// TIA Portal project "Gluing_A1" (V13)

(* hardware
DEVICE "S7300/ET200M-Station_1"  S7-300 station
   slot 0: "Profilschiene_0"  Rail  6ES7 390-1***0-0AA0
   slot 1: "PS 307 5A_1"  PS 307 5A  6ES7 307-1EA00-0AA0
   slot 2: "SIMATIC S7-300"  CPU 314C-2 PN/DP  6ES7 314-6EH04-0AB0  V3.3
      slot 2: "PROFINET-Schnittstelle_1"  PN-IO
         slot 1: "Port_1"  Port
         slot 2: "Port_2"  Port
      slot 5: "DI 24/DO 16_1"  DI24/DO16
      slot 6: "AI 5/AO 2_1"  AI5/AO2
      slot 7: "Zählen_1"  Counter
      slot 8: "Positionieren_1"  Positioning
   slot 4: "CP 343-2_1"  CP 343-2  6GK7 343-2AH01-0XA0  V3.1
*)

// ===== PLC "SIMATIC S7-300"  CPU 314C-2 PN/DP =====

VAR_GLOBAL   // PLC tag table "Standard-Variablentabelle"
   "Ix_S1_Start" AT %I124.0 : Bool;   // Start Pushbutton 1
   "Ix_S2_Start" AT %I124.1 : Bool;   // Start Pushbutton 2
   "Ix_1B1_PressCyl1A1Ret" AT %I124.2 : Bool;   // Press Cylinder 1A1 retracted
   "Ix_1B2_PressCyl1A1Ext" AT %I124.3 : Bool;   // Press Cylinder 1A1 extended
   "Qx_1M1_MovePressCyl1A1Out" AT %Q124.0 : Bool;   // Move PressCylinder 1A1 out
   "Qx_P1_GluingProcess" AT %Q124.7 : Bool;   // Signalise the gluing process
   "Mb_FlagByte10" AT %MB10 : Byte;   // Flag byte 10
   "Mx_Step0" AT %M10.0 : Bool;   // Grafcet, step-flag 0
   "Mx_Step1" AT %M10.1 : Bool;   // Grafcet, step-flag1
   "Mx_Step2" AT %M10.2 : Bool;   // Grafcet, step-flag2
   "Mx_Step3" AT %M10.3 : Bool;   // Grafcet, step-flag3
   "Mx_Step4" AT %M10.4 : Bool;   // Grafcet, step-flag4
   "Mx_Step5" AT %M10.5 : Bool;   // Grafcet, step-flag5
   "Mx_Step6" AT %M10.6 : Bool;   // Grafcet, step-flag6
   "Mx_StartingFlag" AT %M20.0 : Bool;   // Starting flag to activate the sequence (Step 0)
   "Mx_NEdegFlag_Step2" AT %M20.1 : Bool;   // Negative edge flag is activated wehn step 2 is deactivated
   "Mx_Clock10Hz" AT %M100.0 : Bool;   // CPU clock memory-flag 0:f = 10Hz / T=0,1s
   "Mx_Clock5Hz" AT %M100.1 : Bool;   // CPU clock memory-flag 1:f = 5Hz / T=0,2s
   "Mx_Clock2,5Hz" AT %M100.2 : Bool;   // CPU clock memory-flag 2:f = 2,5Hz / T=0,4s
   "Mx_Clock2Hz" AT %M100.3 : Bool;   // CPU clock memory-flag 3:f = 2Hz / T=0,5s
   "Mx_Clock1,2Hz" AT %M100.4 : Bool;   // CPU clock memory-flag 4:f = 1,2Hz / T=0,8s
   "Mx_Clock1Hz" AT %M100.5 : Bool;   // CPU clock memory-flag 5:f = 1Hz / T=1s
   "Mx_Clock0,65Hz" AT %M100.6 : Bool;   // CPU clock memory-flag 6:f = 0,65Hz / T=1,6s
   "Mx_Clock0,5Hz" AT %M100.7 : Bool;   // CPU clock memory-flag 7:f = 0,5Hz / T=2s
   "T_GlueTime" AT %T1 : Timer;   // Adjusting the gluing time
END_VAR

DATA_BLOCK "gluning time value"   // DB2
{ S7_Optimized_Access := 'FALSE' }
VERSION : 0.1
   VAR
      "GluingValue Siemens" : S5Time;
      "GluingValue ICE" : Time;
   END_VAR
BEGIN
END_DATA_BLOCK

FUNCTION "Grafecet" : Void   // FC1, FBD
{ S7_Optimized_Access := 'FALSE' }
VERSION : 0.1
BEGIN

REGION Network 1: step 0
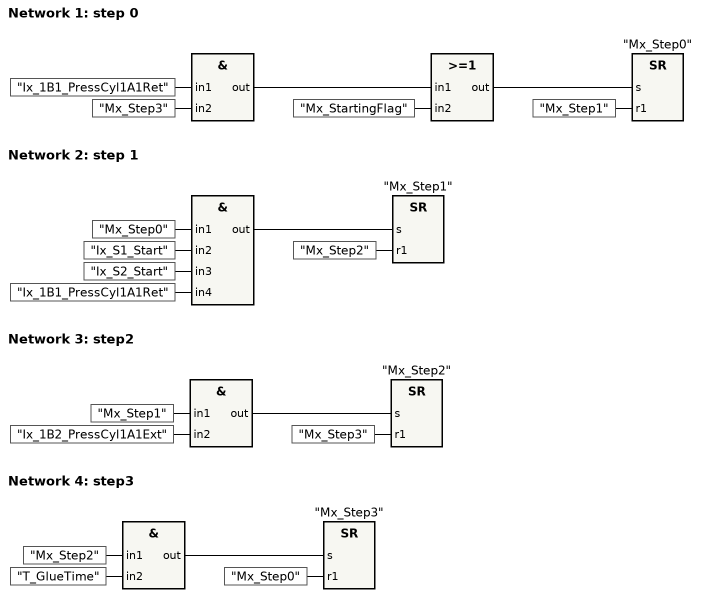
   IF ("Ix_1B1_PressCyl1A1Ret" AND "Mx_Step3") OR "Mx_StartingFlag" THEN
       "Mx_Step0" := TRUE;   // SR flip-flop
   END_IF;
   IF "Mx_Step1" THEN "Mx_Step0" := FALSE; END_IF;
END_REGION

REGION Network 2: step 1
   IF "Mx_Step0" AND "Ix_S1_Start" AND "Ix_S2_Start" AND "Ix_1B1_PressCyl1A1Ret" THEN
       "Mx_Step1" := TRUE;   // SR flip-flop
   END_IF;
   IF "Mx_Step2" THEN "Mx_Step1" := FALSE; END_IF;
END_REGION

REGION Network 3: step2
   IF "Mx_Step1" AND "Ix_1B2_PressCyl1A1Ext" THEN
       "Mx_Step2" := TRUE;   // SR flip-flop
   END_IF;
   IF "Mx_Step3" THEN "Mx_Step2" := FALSE; END_IF;
END_REGION

REGION Network 4: step3
   IF "Mx_Step2" AND "T_GlueTime" THEN
       "Mx_Step3" := TRUE;   // SR flip-flop
   END_IF;
   IF "Mx_Step0" THEN "Mx_Step3" := FALSE; END_IF;
END_REGION
END_FUNCTION

FUNCTION "Actions" : Void   // FC2, FBD
{ S7_Optimized_Access := 'FALSE' }
VERSION : 0.1
BEGIN

REGION Network 1: Set 1M1 1
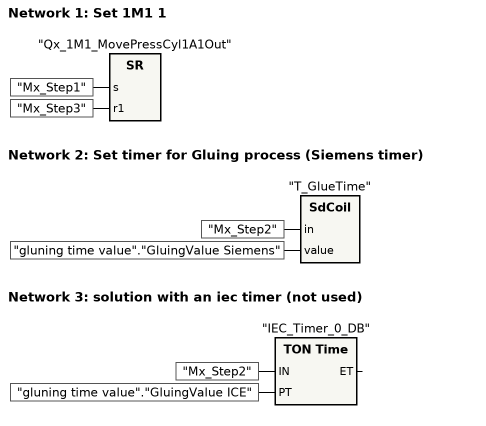
   IF "Mx_Step1" THEN
       "Qx_1M1_MovePressCyl1A1Out" := TRUE;   // SR flip-flop
   END_IF;
   IF "Mx_Step3" THEN "Qx_1M1_MovePressCyl1A1Out" := FALSE; END_IF;
END_REGION

REGION Network 2: Set timer for Gluing process (Siemens timer)
   // no SCL statement known for SdCoil: written as a call
   SdCoil(in := "Mx_Step2", value := "gluning time value"."GluingValue Siemens", operand := "T_GlueTime");
END_REGION

REGION Network 3: solution with an iec timer (not used)
   "IEC_Timer_0_DB".TON(IN := "Mx_Step2", PT := "gluning time value"."GluingValue ICE");
END_REGION
END_FUNCTION

ORGANIZATION_BLOCK "Main"   // OB1, FBD
TITLE = "Main Program Sweep (Cycle)"
{ S7_Optimized_Access := 'FALSE' }
VERSION : 0.1
BEGIN

REGION Network 1
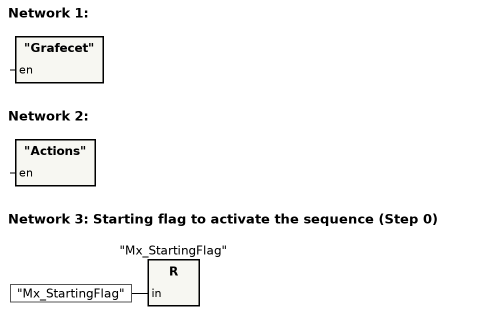
   "Grafecet"();
END_REGION

REGION Network 2
   "Actions"();
END_REGION

REGION Network 3: Starting flag to activate the sequence (Step 0)
   IF "Mx_StartingFlag" THEN "Mx_StartingFlag" := FALSE; END_IF;
END_REGION
END_ORGANIZATION_BLOCK

ORGANIZATION_BLOCK "COMPLETE RESTART"   // OB100, FBD
TITLE = "Complete Restart"
{ S7_Optimized_Access := 'FALSE' }
VERSION : 0.1
BEGIN

REGION Network 1: Flag byte 10
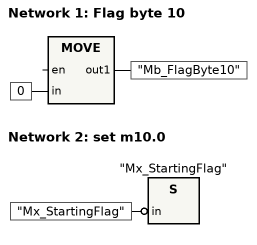
   "Mb_FlagByte10" := 0;
END_REGION

REGION Network 2: set m10.0
   IF NOT "Mx_StartingFlag" THEN "Mx_StartingFlag" := TRUE; END_IF;
END_REGION
END_ORGANIZATION_BLOCK